{attribute addProperty BoxType "EL2521-0124-0016"}
{attribute addProperty Id "PTO_StatusAT %I*PTO_Status_C602A91E4050ENC_Status_compactAT %I*ENC_Status_compact_3D845C6988110PLS_StatusAT %I*PLS_Status_B10359913240PTO_ControlAT %Q*PTO_Control_DFE022934050ENC_Control_compactAT %Q*ENC_Control_compact_14754A394050PLS_Control_compactAT %Q*PLS_Control_compact_12AF77AA4860WcStateAT %I*WcState_98A4DF7520.250InfoDataAT %I*InfoData_BC63D37F80100"}
{attribute addProperty CRC "4114602728"}
{attribute addProperty SizeInBites "370"}
{attribute addProperty SizeInBytes "46.25"}
TYPE EL2521_8CF885D4 :
STRUCT
	{attribute addProperty Name "PTO_Status"}
	PTO_Status : PTO_Status_C602A91E;
	{attribute addProperty Name "ENC_Status_compact"}
	ENC_Status_compact : ENC_Status_compact_3D845C69;
	{attribute addProperty Name "PLS_Status"}
	PLS_Status : PLS_Status_B1035991;
	{attribute addProperty Name "PTO_Control"}
	PTO_Control : PTO_Control_DFE02293;
	{attribute addProperty Name "ENC_Control_compact"}
	ENC_Control_compact : ENC_Control_compact_14754A39;
	{attribute addProperty Name "PLS_Control_compact"}
	PLS_Control_compact : PLS_Control_compact_12AF77AA;
	{attribute addProperty Name "WcState"}
	WcState : WcState_98A4DF75;
	{attribute addProperty Name "InfoData"}
	InfoData : InfoData_BC63D37F;
END_STRUCT
END_TYPE

(* stored: Version 1.2.0.0, ProductVersion 3.1.4024.9
   DUT EL2521_8CF885D4: Id {109019d3-4384-4e54-bf47-bf0e4f5723bd} *)
